// TIA Portal V17 export
// export: Created 2022-07-28T18:03:17.2577632Z, ExportSetting None, DisplayName Totally Integrated Automation Portal, DisplayVersion V17, DisplayName TIA Portal Openness, DisplayVersion V17, DisplayName TIA Portal Teamcenter Gateway, DisplayVersion V17, DisplayName TIA Portal Version Control Interface, DisplayVersion V17, DisplayName TIA Portal Test Suite Advanced, DisplayVersion V17, DisplayName SINAMICS Startdrive Advanced, DisplayVersion V17, DisplayName SINAMICS DCC, DisplayVersion V17, DisplayName SINAMICS Startdrive G130, G150, S120, S150, SINAMICS MV, S210, DisplayVersion V17, DisplayName SINAMICS Startdrive G110M, G120, G120C, G120D, G120P, G115D, DisplayVersion V17, DisplayName STEP 7 Professional, DisplayVersion V17, DisplayName SIMATIC Energy Suite, DisplayVersion V17, DisplayName STEP 7 CFC, DisplayVersion V17, DisplayName STEP 7 Safety, DisplayVersion V17, DisplayName WinCC Advanced / Unified PC, DisplayVersion V17, DisplayName SIMATIC Visualization Architect, DisplayVersion V17
TYPE "_Inverter_352Tel_Send"
   STRUCT
      CTW : "_Inverter_352Tel_CTW_Bits";   // Control word
      r_ReferenceSpeed : Real := 100.0;   // Reference speed, P2000
      r_ReferenceCurrent : Real := 100.0;   // Reference current, P2002
      r_ReferenceTorque : Real := 100.0;   // Reference torque, P2003
      r_SetpointSpeed : Real;   // Setpoint speed, %. Negative value change direction.
   END_STRUCT;
END_TYPE
